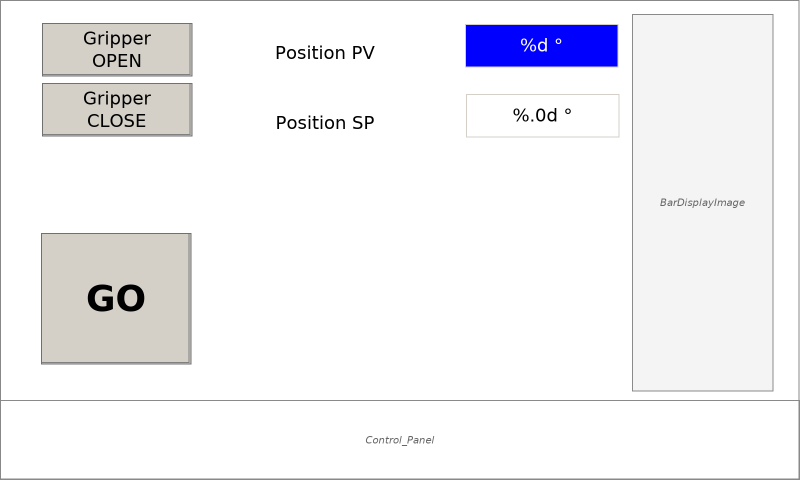
VISUALIZATION Servo  // 800x480
    Frame (0,400 800x80)
        shows Control_Panel()
    BarDisplayImage (632,14 141x377), value: ServoCtrl.ActualCurrent, style: BarDisplayImage-Gray, scale format: %.0d, scale 0..2000
        p518627256: Motor I, Amper
    Textfield (466,94 153x43), "%.0d °", text variable: GVL_IO.Position_SP
        OnMouseClick: write the text variable via Default
    Button (41,233 150x131), "GO"
        tap GVL_IO.GO_TO_cmd
    Label (250,38 150x30), "Position PV"
    Label (250,108 150x30), "Position SP"
    Textfield (465,24 153x43), "%d °", text variable: GVL_IO.Position_PV_HMI
    Button (42,23 150x53), "Gripper OPEN", colour toggle: GVL_IO.ixGripper_Unlock
        tap GVL_IO.Gripper_Open_cmd
    Button (42,83 150x53), "Gripper CLOSE", colour toggle: GVL_IO.TwoSensorLock
        tap GVL_IO.Gripper_Close_cmd
END_VISUALIZATION

(* stored: Version 1.1.0.1, ProductVersion 3.1.4024.13
   Visu Servo: Id {c75d5d9a-7be5-4d4b-9dc3-5429ff94ea9b} *)
